// Core §6.9(b) — named plain-condition wait
TYPE ST_CondRecord :
STRUCT
    Label : STRING(120);   // localization key
    Ok    : BOOL;
END_STRUCT
END_TYPE

(* stored: Version 1.1.0.1, ProductVersion 3.1.4024.12
   DUT ST_CondRecord: Id {4ba68801-ca97-4872-9555-2ff4a8f36dce} *)
